(* CoDeSys 2.3 library: TcCX1000System.lib *)
(* Libraries: STANDARD.LIB*5.6.98 12:03:02, TcBase.lib*14.5.09 12:14:08, TcSystem.lib*9.3.10 11:21:30 *)

(* Global variable list: Global_Constants *)
VAR_GLOBAL CONSTANT
(* ===============================	*)
(* Definition globaler Konstanten			*)
(* ===============================	*)
	iLength	:	INT := 40;


	IOADS_IGR_IODEVICESTATE_BASE : INT :=		16#00005000;	(* plus ID des jeweiligen Device *)





END_VAR

(* Data type *)
TYPE
	E_CX1000_DisplayModes :
	(
		e_CX1000_DisplayNoAction := 0,
		e_CX1000_DisplayOn		:= 1,
		e_CX1000_DisplayOff,
		e_CX1000_CursorOn,
		e_CX1000_CursorOff,
		e_CX1000_CursorBlinkOn,
		e_CX1000_CursorBlinkOff,
		e_CX1000_BackLightOn,
		e_CX1000_BackLightOff,
		e_CX1000_ClearDisplay,
		e_CX1000_WriteLine1,
		e_CX1000_WriteLine2
	);
END_TYPE

(* Data type *)
TYPE E_UPS_STATE : (
	eUPS_UNDEF,
	eUPS_CHARGING,
	eUPS_CHARGED,
	eUPS_DISCHARGE,
	eUPS_DISCHARGE_RESTART,
	eUPS_OUTPUT_OFF,
	eUPS_OVERLOAD
);
END_TYPE

(* Data type *)
TYPE ST_CX1000_ProfilerStruct :
STRUCT
	dwLastExecTime		: DWORD;
	dwMinExecTime		: DWORD;
	dwMaxExecTime		: DWORD;
	dwAverageExecTime	: DWORD;
	dwMeasureCycle		: DWORD;
END_STRUCT
END_TYPE

(* POU F_CX1000SetWatchdog, ST *)
FUNCTION F_CX1000SetWatchdog : BOOL
VAR_INPUT
	tTimeOut		: TIME; 			(* Watchdog TimeOut Time *)
	bEnable			: BOOL; 			(* Enable / Disable Watchdog *)
END_VAR
VAR
	nValue			: DWORD;
END_VAR
VAR CONSTANT
	nPortAddr		: UDINT := 16#9000;
	nWDConfig		: DWORD := 2#00000001_11110101_00000000_00000000;
(*
	TimerScale = 32kHz / (2^nWDPreScaler)

						 -----WDCNFG------ ------WDTO------ 
	WD32KhzEnable	= 2#00000001_00000000_00000000_00000000  // Enable Watchdog 32 kHz Clock
	WDEventType2	= 2#00000000_11000000_00000000_00000000  // Watchdog event type 2 (System Reset)
	WDEventType1	= 2#00000000_00110000_00000000_00000000  // Watchdog event type 1 (System Reset)
	WDPreScaler		= 2#00000000_00000101_00000000_00000000  // Watchdog Prescaler (Divide 32kHz by 32)
*)
END_VAR
IF bEnable THEN
	(* watchdog active *)
	nValue			  	:= nWDConfig OR ((TIME_TO_DWORD(tTimeOut)) AND 16#0000FFFF);
	F_CX1000SetWatchdog := FW_PortWrite (nPortAddr, SIZEOF(nValue), nValue);
ELSE
	(* watchdog deactivated *)
	nValue			  	:= nWDConfig AND 16#FFFF0000;
	F_CX1000SetWatchdog := FW_PortWrite (nPortAddr, SIZEOF(nValue), nValue);
END_IF
END_FUNCTION

(* POU F_CX1000SubTimeStamp, ST *)
(* Calculates "TimeStamp_A" minus "TimeStamp_B" and returns the resulting time difference
		as "F_CX1000SubTimeStamp" in microseconds 

 IN:	TimeStamp_A		(2 x UDINT)		[100*ns]										
		TimeStamp_B		(2 x UDINT)		[100*ns]										

 OUT:	TimeDifference	(1 x UDINT)	[us] limited to 0..4294967295us (16#FFFFFFFF)	
		negative and huge differences are returned as 4294967295us (71m34s967ms295us)	
		in case of negative or huge differences use UInt64Sub64() of TcUtilities.lib 	*)

FUNCTION F_CX1000SubTimeStamp : UDINT		(* [us] *)
VAR_INPUT
	nTimeStampLoDW_A	: UDINT;	(* 2*32 bit time stamp A: low DWORD					*)
	nTimeStampHiDW_A	: UDINT;	(* 2*32 bit time stamp A: high DWORD				*)
	nTimeStampLoDW_B	: UDINT;	(* 2*32 bit time stamp B: low DWORD					*)
	nTimeStampHiDW_B	: UDINT;	(* 2*32 bit time stamp B: high DWORD				*)
END_VAR
VAR
	nDeltaTimeStampLoDW	: UDINT;	(* 2*32 bit delta time stamp for low DWORD			*)
	nDeltaTimeStampHiDW	: UDINT;	(* 2*32 bit delta time stamp for high DWORD			*)
END_VAR
VAR CONSTANT
	fSCALE_LOWDW		: LREAL	:= 0.1;	(* time stamp in [100*ns]: 1=0.1 us (1.0 / 10.0)*)
	fSCALE_HIGHDW		: LREAL := 429496729.6;	(* 4294967296(2^32) / 10				*)
END_VAR
(* calculate time difference per DWORD *)
nDeltaTimeStampLoDW := nTimeStampLoDW_A - nTimeStampLoDW_B;
nDeltaTimeStampHiDW := nTimeStampHiDW_A - nTimeStampHiDW_B;

IF ( nTimeStampLoDW_A >= nTimeStampLoDW_B ) THEN
	F_CX1000SubTimeStamp	:= LREAL_TO_UDINT(
		LIMIT(
			0,
			UDINT_TO_LREAL(nDeltaTimeStampHiDW) * 429496729.6 + UDINT_TO_LREAL(nDeltaTimeStampLoDW) / 10.0,
			4294967295)
	);
ELSE
	F_CX1000SubTimeStamp	:= LREAL_TO_UDINT(
		LIMIT(
			0,
			UDINT_TO_LREAL(nDeltaTimeStampHiDW - 1) * 429496729.6 + UDINT_TO_LREAL(nDeltaTimeStampLoDW) / 10.0,
			4294967295)
	);
END_IF;
END_FUNCTION

(* POU F_GetVersionTcCX1000System, ST *)
FUNCTION F_GetVersionTcCX1000System : UINT
VAR_INPUT
	nVersionElement		:	INT;
END_VAR
(*
	Possible nVersionElement parameter:
	1	:	major number
	2	:	minor number
	3	:	revision number
*)
VAR
END_VAR
(* Version history:
Date			| Version			| created under							| Author					| Remark 
------------------------------------------------------------------------------------------------------------------------------------------------------------------------------------------------------------------------------------------ 
2005/10/05    	| 1.0.1				| V2.10.0 (Build 1242)						| ICh						| UPS-FBs are now using ADSSTATE_POWERFAILURE to stop WinCE/XP, 
2005/10/05    	| 1.0.1				| V2.10.0 (Build 1242)						| ICh						| F_GetVersionTcCX1000System added 
2007/01/29    	| 1.0.2				| V2.10.0 (Build 1307)						| ICh						| Fix for large and negative differences in F_CX1000SubTimeStamp, fix for FB_CX1000SimpleUps 
11.10.2010	| 1.0.3				| TCAT2.11 B2015							| Christoph C				| Small correction in the FB_CX1000Profiler function block (calculation of average velue for a first measure cycle )
*) 
CASE nVersionElement OF
1:	(* major number *)
	F_GetVersionTcCX1000System := 1;
2:	(* minor number *)
	F_GetVersionTcCX1000System := 0;
3:	(* revision number *)
	F_GetVersionTcCX1000System := 3;
ELSE
	F_GetVersionTcCX1000System := 16#FFFF;
END_CASE
END_FUNCTION

(* POU FB_CX1000Profiler, ST *)
FUNCTION_BLOCK FB_CX1000Profiler
VAR_INPUT
	bStart					: BOOL;(*rising edge starts measurement and falling stops*)
	bReset					: BOOL;
END_VAR
VAR_OUTPUT
	bBusy					: BOOL;
	stData					: ST_CX1000_ProfilerStruct;
END_VAR
VAR CONSTANT
	iMAX_DATABUFF_SIZE		: INT := 100;
	iMAX_AVERAGE_MEASURES 	: INT := 100;
END_VAR
VAR
	fbRisingEdgeStart		: R_TRIG;
	fbRisingEdgeReset		: R_TRIG;
	fbFallingEdgeStart		: F_TRIG;
	fbGetCPUCounter			: GETCPUCOUNTER;
	dwOldCpuCntLo			: DWORD:=0;
	dwOldCpuCntHi			: DWORD:=0;
	dwOldCpuCntDiff			: DWORD:=0;
	dwNewCpuCntLo			: DWORD:=0;
	dwNewCpuCntHi			: DWORD:=0;
	dwNewCpuCntDiff		: DWORD:=0;
	aMeasureData			: ARRAY[0..iMAX_DATABUFF_SIZE] OF DWORD;
	dwTimeSum				: DWORD:=0;
	iMaxData					: INT:=1;
	iIdx							: DWORD:=0;
END_VAR
fbFallingEdgeStart(CLK:=bStart);

IF ( fbFallingEdgeStart.Q ) THEN
	fbGetCPUCounter();	(*get current counter value*)
	dwNewCpuCntLo := fbGetCPUCounter.cpuCntLoDW;
	dwNewCpuCntHi := fbGetCPUCounter.cpuCntHiDW;

	dwNewCpuCntDiff := F_CX1000SubTimeStamp(dwNewCpuCntLo, dwNewCpuCntHi, dwOldCpuCntLo, dwOldCpuCntHi);

	stData.dwLastExecTime	:=	 dwNewCpuCntDiff; (* in us *)

	(*calculate the min and max*)
	IF ( stData.dwMeasureCycle = 1 ) THEN  			(*first measurement*)
		stData.dwMinExecTime 	:= 	stData.dwLastExecTime;
		stData.dwMaxExecTime 	:= 	stData.dwLastExecTime;
	ELSE	(* ( Overflow->stData.MeasureCycle==0 ) or ( measure > 1 ) *)
		stData.dwMinExecTime 	:=	MIN( stData.dwMinExecTime, stData.dwLastExecTime );
		stData.dwMaxExecTime 	:=	MAX( stData.dwMaxExecTime, stData.dwLastExecTime );
	END_IF

	(* save last value to the data buffer *)
	aMeasureData[ stData.dwMeasureCycle MOD iMaxData  (*0..iMaxData - 1*)]	:= 	stData.dwLastExecTime;

	(*calculate average values*)
	dwTimeSum	:= 0;
	IF ( stData.dwMeasureCycle >= iMaxData ) OR  ( stData.dwMeasureCycle = 0 ) THEN (*add all values*)
		FOR iIdx := 0 TO ( iMaxData - 1 ) DO
			dwTimeSum 	:= 	dwTimeSum + aMeasureData[ iIdx ];
		END_FOR
		stData.dwAverageExecTime	:= 	dwTimeSum / iMaxData;
	ELSE
		FOR  iIdx:=1  TO stData.dwMeasureCycle DO
			dwTimeSum 	:= 	dwTimeSum + aMeasureData[ iIdx ];
		END_FOR
		stData.dwAverageExecTime	:= 	dwTimeSum / stData.dwMeasureCycle;
	END_IF

	bBusy:=FALSE;
END_IF


fbRisingEdgeStart(CLK:=bStart);
fbRisingEdgeReset(CLK:=bReset);
IF ( fbRisingEdgeStart.Q ) THEN
	bBusy:=TRUE;

	IF ( fbRisingEdgeReset.Q ) THEN
		stData.dwLastExecTime := 0;
		stData.dwMinExecTime := 0;
		stData.dwMaxExecTime := 0;
		stData.dwAverageExecTime:=0;
		stData.dwMeasureCycle:=0;
		dwTimeSum := 0;
		FOR iIdx := 0 TO iMaxData DO
			aMeasureData[ iIdx ]:=0;	(*clear buffer*)
		END_FOR;
	END_IF

	iMaxData:= MAX( 2, MIN( iMAX_DATABUFF_SIZE,  iMAX_AVERAGE_MEASURES ) );
	stData.dwMeasureCycle	:=	stData.dwMeasureCycle + 1;		(*increment measure cycle counter*)

	fbGetCPUCounter();								(*get current counter value*)
													(* save start  value*)
	dwOldCpuCntLo := fbGetCPUCounter.cpuCntLoDW;
	dwOldCpuCntHi := fbGetCPUCounter.cpuCntHiDW;
END_IF
END_FUNCTION_BLOCK

(* POU FB_CX1000SetTextDisplay, ST *)
FUNCTION_BLOCK FB_CX1000SetTextDisplay
VAR_INPUT
	bExecute : BOOL;
	nDevID	:	UDINT;
	nMode	: E_CX1000_DisplayModes;
	stLine : STRING(20);
	nCursorPos : DWORD;
END_VAR
VAR_OUTPUT
	bBusy : BOOL;
	bErr	:	BOOL;
	nErrorID	:	UDINT;
END_VAR
VAR
	step : INT := 100;
	fbADSWrite : ADSWRITE;
	bStarted : BOOL;
	nIndexOffset : UDINT;
	nWriteMode : INT;
	fbOnTrigger		:	R_TRIG;
	temp : DWORD;
END_VAR
VAR CONSTANT
	(* write mode *)
	WRITE_MODE_IDLE	: INT := 1;
	WRITE_MODE_BYTE	: INT := 2;
	WRITE_MODE_STRING	: INT := 3;

	(*  CX1100 *)
	IOADS_IOF_CX1100_WRITE1LINE : UDINT :=		16#FFFF00FF;
	IOADS_IOF_CX1100_WRITE2LINE : UDINT :=		16#FFFF40FF;
	IOADS_IOF_CX1100_WRITECURSOR : UDINT :=		16#FFFF80FF;
	IOADS_IOF_CX1100_FILLRAW : UDINT :=		16#FFFF81FF;
	IOADS_IOF_CX1100_CURSOR_OFF : UDINT :=		16#FFFF90FF;
	IOADS_IOF_CX1100_CURSOR_ON : UDINT :=		16#FFFF91FF;
	IOADS_IOF_CX1100_CURSOR_BOFF : UDINT :=		16#FFFF92FF;
	IOADS_IOF_CX1100_CURSOR_BON : UDINT :=		16#FFFF93FF;
	IOADS_IOF_CX1100_DISPLAY_OFF : UDINT :=		16#FFFF94FF;
	IOADS_IOF_CX1100_DISPLAY_ON : UDINT :=		16#FFFF95FF;
	IOADS_IOF_CX1100_BACKLIGHT_ON : UDINT :=		16#FFFF96FF;
	IOADS_IOF_CX1100_BACKLIGHT_OFF : UDINT :=		16#FFFF97FF;
	IOADS_IOF_CX1100_CLEARDISPLAY : UDINT :=		16#FFFFA0FF;

	IOADS_IOF_CX1100_TERMTYPES : UDINT :=		16#FFFF0001;
END_VAR
CASE step OF
100 :
	fbOnTrigger(CLK:= bExecute);
    	IF fbOnTrigger.Q OR bStarted
	THEN
		bStarted := TRUE;
		bBusy := TRUE;
		bErr := FALSE;
		nErrorID := 0;
		(* select action *)
		CASE nMode OF
			e_CX1000_DisplayNoAction:
				nIndexOffset := 0;
				nWriteMode := WRITE_MODE_IDLE;
			e_CX1000_DisplayOn:
				nIndexOffset := IOADS_IOF_CX1100_DISPLAY_ON;
				nWriteMode := WRITE_MODE_BYTE;
			e_CX1000_DisplayOff:
				nIndexOffset := IOADS_IOF_CX1100_DISPLAY_OFF;
				nWriteMode := WRITE_MODE_BYTE;
			e_CX1000_CursorOn:
				nIndexOffset := IOADS_IOF_CX1100_CURSOR_ON;
				nWriteMode := WRITE_MODE_BYTE;
			e_CX1000_CursorOff:
				nIndexOffset := IOADS_IOF_CX1100_CURSOR_ON;
				nWriteMode := WRITE_MODE_BYTE;
			e_CX1000_CursorBlinkOn:
				nIndexOffset := IOADS_IOF_CX1100_CURSOR_BON;
				nWriteMode := WRITE_MODE_BYTE;
			e_CX1000_CursorBlinkOff:
				nIndexOffset := IOADS_IOF_CX1100_CURSOR_BOFF;
				nWriteMode := WRITE_MODE_BYTE;
			e_CX1000_BackLightOn:
				nIndexOffset := IOADS_IOF_CX1100_BACKLIGHT_ON;
				nWriteMode := WRITE_MODE_BYTE;
			e_CX1000_BackLightOff:
				nIndexOffset := IOADS_IOF_CX1100_BACKLIGHT_OFF;
				nWriteMode := WRITE_MODE_BYTE;
			e_CX1000_ClearDisplay:
				nIndexOffset := IOADS_IOF_CX1100_CLEARDISPLAY;
				nWriteMode := WRITE_MODE_BYTE;
			e_CX1000_WriteLine1:
				IF nCursorPos <> 0
				THEN
					IF nCursorPos < 15
					THEN
						nIndexOffset := DWORD_TO_UDINT( UDINT_TO_DWORD(IOADS_IOF_CX1100_WRITE1LINE) OR (SHL(nCursorPos,8)));
					ELSE
						nIndexOffset := 0;
						nWriteMode := WRITE_MODE_IDLE;
						bErr := TRUE;
						nErrorID := 4711;
					END_IF;
				ELSE
					nIndexOffset := IOADS_IOF_CX1100_WRITE1LINE;
				END_IF;
				nWriteMode := WRITE_MODE_STRING;
			e_CX1000_WriteLine2:
				IF nCursorPos <> 0
				THEN
					IF nCursorPos < 15
					THEN
						nIndexOffset := DWORD_TO_UDINT( UDINT_TO_DWORD(IOADS_IOF_CX1100_WRITE2LINE) OR (SHL(nCursorPos,8)));
					ELSE
						nIndexOffset := 0;
						nWriteMode := WRITE_MODE_IDLE;
						bErr := TRUE;
						nErrorID := 4711;
					END_IF;
				ELSE
					nIndexOffset := IOADS_IOF_CX1100_WRITE2LINE;
				END_IF;
				nWriteMode := WRITE_MODE_STRING;
		ELSE
			;
		END_CASE;
		CASE nWriteMode OF
			WRITE_MODE_IDLE :
				;
			WRITE_MODE_BYTE:
				fbADSWrite(NETID:= '',
					PORT:= 300,
					IDXGRP:= 16#5000+nDevID,
					IDXOFFS:= nIndexOffset,
					LEN:= 0,
					SRCADDR:= 0,
					WRITE:= TRUE,
					TMOUT:= t#1s);
			WRITE_MODE_STRING:
				fbADSWrite(NETID:= '',
					PORT:= 300,
					IDXGRP:= 16#5000+nDevID,
					IDXOFFS:= nIndexOffset,
					LEN:= LEN(stLine),
					SRCADDR:= ADR(stLine),
					WRITE:= TRUE,
					TMOUT:= t#1s);
		END_CASE;

		IF NOT fbADSWrite.BUSY OR (nWriteMode = WRITE_MODE_IDLE)
		THEN
			bStarted := FALSE;
			step := 300;
		END_IF;
	END_IF;
300:
	IF NOT fbADSWrite.err
	THEN
		step := 100;
	ELSE
		bErr := TRUE;
		nErrorID := fbADSWrite.ERRID;
		step := 100;
	END_IF;
	fbADSWrite( WRITE:= FALSE );
	bBusy := FALSE;
END_CASE;
END_FUNCTION_BLOCK

(* POU FB_CX1000SimpleUps, ST *)
FUNCTION_BLOCK FB_CX1000SimpleUps
VAR_INPUT
	bDIPDisable			: BOOL;	(* If TRUE override Dip Switch *)
	iDischargeLevel		: USINT;(* Discharge Switch Off Level: 0 = 100%, 9 = 90%, 8 = 80%, ..., 2 = 20%, 1 = 10% *)
	tDelay				: TIME;	(* Time to hold during power failure (shutdown after timer ellapses) [0s .. 10s] *)
END_VAR
VAR_OUTPUT
	bPowerFailure		: BOOL;	(* True if power fault detected *)
	bShutdownActive		: BOOL;	(* True if shutdown is actively executed *)
	bUpsReady			: BOOL;	(* True if UPS 24V Out is OK *)
	b24VInOK			: BOOL;	(* True if UPS 24V In is OK *)
	bHolding			: BOOL;	(* True if power fault detected and tDelay not yet ellapsed *)
	tTimeUntilShutdown	: TIME;	(* Remaining Time until system shuts down during power failure *)
	eUpsState			: E_UPS_STATE; (* UPS-State [UNDEF | CHARGING | CHARGED | DISCHARGE |
													 DISCHARGE_RESTART | OUTPUT_OFF | OVERLOAD] *)
END_VAR
VAR
	Ii24VState AT %I* 	: BYTE;
	IiChargeState AT %I*: BYTE;
	QiControl AT %Q*	: BYTE;
	QiDipControl AT %Q*	: BYTE;

	iState				: INT := 0; (* 0: IDLE, 1: HOLDING, 2: SHUTDOWN *)
	HoldTimer			: TON;
	fbShutdown			: ADSWRTCTL;  (* Windows shutdown *)
	dwDelay				: DWORD := 0; (* 0 immediate shutdown of Windows, [s] *)
	WaitStateTime		: TON;		(*Wait for state UPS*)
	bEndOfHolding		: BOOL;		(*Phase before Shutdown activ*)
END_VAR
VAR CONSTANT
	tWaitStateTime		: TIME := t#2s500ms;
END_VAR
(* status *)
b24VInOK		:= Ii24VState.1;
bUpsReady		:= Ii24VState.0;
bPowerFailure 	:= NOT(Ii24VState.1);
eUpsState		:= SHR((Ii24VState AND 16#F0), 4);
QiControl.2 	:= bDIPDisable;

(* limit holding time *)
IF tDelay > T#10s THEN
	tDelay := T#10s;
END_IF

HoldTimer(PT := tDelay, IN := bPowerFailure);
WaitStateTime(PT := tWaitStateTime, IN := bEndOfHolding);

(* override DIP switch with iDischargeLevel *)
IF bDIPDisable THEN
	IF iDischargeLevel > 9 THEN  (* limit SW Dip Switch *)
		QiDipControl := 0;
	ELSE
		QiDipControl := iDischargeLevel;
	END_IF
END_IF

CASE iState OF
0: (* IDLE *)
	(* make sure link to IiChargeState exists (assume link to Ii24VState is then also there) before evaluating power failure to avoid constant reboot *)
	IF bPowerFailure AND (eUpsState <> eUPS_UNDEF) THEN
		QiControl.3 := TRUE; (* set auto reset while holding *)
		iState 		:= 1;
	END_IF

1: (* HOLD *)
	IF b24VInOK THEN
		(* power failure has ended before hold timer ellapsed *)
		QiControl.3 := FALSE; (* clear auto reset *)
		iState 		:= 0;

	ELSIF HoldTimer.Q THEN
		(* power failure has continued until hold timer ellapsed *)
		bEndOfHolding	:= TRUE;
		QiControl.3 	:= FALSE; (* clear auto reset *)
		iState 			:= 2;
	END_IF

2: (* Wait for state UPS *)
	IF WaitStateTime.Q  THEN
		bEndOfHolding	:= FALSE;
		IF (eUpsState=eUPS_CHARGED) OR (eUpsState=eUPS_CHARGING)THEN
			(* no shutdown required since CX power supply is not discharging *)
			iState := 0;
		ELSE
			bShutdownActive := TRUE;
			fbShutdown(
				NETID 		:= '',
				PORT 		:= AMSPORT_R3_SYSSERV,
				ADSSTATE 	:= ADSSTATE_POWERFAILURE, (* Windows Shutdown *)
				DEVSTATE 	:= 0,
				LEN 		:= SIZEOF(dwDelay),
				SRCADDR 	:= ADR(dwDelay),
				Write 		:= TRUE,
				TMOUT 	:= T#3s
			);
			iState 			:= 3;
		END_IF
	END_IF

3: (* SHUTDOWN *)
	fbShutdown(Write := TRUE);
END_CASE

(* status *)
bHolding 			:= QiControl.3;
tTimeUntilShutdown	:= HoldTimer.PT - HoldTimer.ET;
END_FUNCTION_BLOCK

(* POU FB_CX1000UpsHandling, ST *)
FUNCTION_BLOCK FB_CX1000UpsHandling
VAR_INPUT
	bAutoReset				: BOOL; (* if True, keep CX1000 alive if power is restored *)
	bDIPDisable				: BOOL; (* if True, overwrite DIP settings (rotary switch) *)
	bShutdown24V			: BOOL;	(* switch off 24V *)
	bShutdown5V				: BOOL; (* switch off  5V *)
	iDischargeLevel			: USINT;(* UPS switches off if 10, 20, .. 100[%] charge level is discharged *)
	bTcStopOnly				: BOOL; (* TwinCAT stop instead of Windows Shutdown *)
	tDelay					: TIME;	(* delay time before stop/shutdown *)
END_VAR
VAR_OUTPUT
	bPowerFailure			: BOOL;	(* True if power fault detected *)
	bShutdownActive			: BOOL;	(* True if shutdown is actively executed *)
	bUpsReady				: BOOL;	(* True if UPS 24V Out is OK *)
	b24VInOK				: BOOL;	(* True if UPS 24V In is OK *)
END_VAR
VAR
	(* to be linked in System Manager with I/O from CX1100|CX1190-UPS *)
	Ii24VState AT %I*		: BYTE;
	IiChargeState AT %I*	: USINT;
	QiControl AT %Q*		: BYTE;
	QiDIPControl AT %Q*		: USINT;

	(* ups powerfault detection via wired digital input from UPS Power Connector *)
	IbPowerFault	AT %I*	: BOOL;

	(* edge detection *)
	b24VInOKPrev			: BOOL;
	bPowerFaultPrev			: BOOL;
	(*iIRQ					: BYTE;*)(* IRQ 0..3 *)

	(* powerfault reaction *)
	PowerFailTimer			: TON;		  (* holding timer *)
	dwDelay					: DWORD := 0; (* 0 immediate shutdown of Windows, [s] *)
	bPowerFaultInit			: BOOL  := TRUE;
	fbPowerFaultReaction	: ADSWRTCTL;  (* TwinCAT Stop or Windows shutdown *)
END_VAR
(* Status *)
b24VInOK	:= Ii24VState.1;
bUpsReady	:= Ii24VState.0;

(* Control *)
QiControl	:= 16#00;
QiControl.0 := bShutdown5V;
QiControl.1 := bShutdown24V;
QiControl.2 := bDIPDisable;
QiControl.3 := bAutoReset;

(*
CASE LIMIT(0, iIRQ, 3) OF
	0:	QiControl.4 := TRUE;
	1:	QiControl.5 := TRUE;
	2:	QiControl.6 := TRUE;
	3:	QiControl.7 := TRUE;
END_CASE
*)

(* DIP 1 = 10%, DIP 2 = 20%, .. DIP 9 = 90%, DIP 0 = 100% *)
QiDIPControl := LIMIT(0, iDischargeLevel/10 MOD 10, 10);

IF ((NOT(b24VInOK) AND b24VInOKPrev) OR (IbPowerFault AND NOT(bPowerFaultPrev)))
	AND NOT(bShutdownActive) THEN

	(* set shutdown request on rising edge of input 24V power fault detection *)
	bPowerFailure 		:= TRUE;
	bPowerFaultInit		:= TRUE;
ELSIF ((b24VInOK AND NOT(b24VInOKPrev)) OR (NOT(IbPowerFault) AND bPowerFaultPrev))
	AND bAutoReset THEN

	(* reset shutdown request on falling edge of input 24V power fault detection *)
	bPowerFailure 	:= FALSE;
	bPowerFaultInit	:= TRUE;
END_IF

(* holding time *)
PowerFailTimer(PT := tDelay, IN := bPowerFailure);

IF PowerFailTimer.Q OR bShutdownActive THEN
	(* shutdown requested, acknowledged and holding time expired - execute shutdown *)
	IF bPowerFaultInit THEN
		bPowerFaultInit := FALSE;
		bShutdownActive	:= TRUE;

		IF bTcStopOnly THEN
			fbPowerFaultReaction(Write := FALSE);
			fbPowerFaultReaction(
				NETID 	 	:= '',
				PORT 	 	:= AMSPORT_R3_SYSSERV,
				ADSSTATE 	:= ADSSTATE_STOP, 	 (* TwinCAT Stop *)
				DEVSTATE 	:= 0,
				LEN 	 	:= 0,
				SRCADDR  	:= 0,
				Write 	 	:= TRUE,
				TMOUT 	 	:= T#3s
			);
		ELSE
			fbPowerFaultReaction(Write := FALSE);
			fbPowerFaultReaction(
				NETID 		:= '',
				PORT 		:= AMSPORT_R3_SYSSERV,
				ADSSTATE 	:= ADSSTATE_POWERFAILURE, (* Windows Shutdown *)
				DEVSTATE 	:= 0,
				LEN 		:= SIZEOF(dwDelay),
				SRCADDR 	:= ADR(dwDelay),
				Write 		:= TRUE,
				TMOUT 		:= T#3s
			);
		END_IF
	ELSE
		fbPowerFaultReaction(Write := FALSE);

		IF NOT(fbPowerFaultReaction.BUSY) THEN
			fbPowerFaultReaction(Write := FALSE);
			bPowerFailure := FALSE;
		END_IF
	END_IF
END_IF

b24VInOKPrev	:= b24VInOK;
bPowerFaultPrev := IbPowerFault;
END_FUNCTION_BLOCK
